// TIA Portal V21 export
FUNCTION "T_PausaLavoro" : Void   // FC81, LAD
{ S7_Optimized_Access := 'TRUE' }
// stored: SetENOAutomatically false
   VAR_IN_OUT
      PausaLavoro : "Std_PausaLavoro";
   END_VAR
   VAR_TEMP   // added for the SCL form of the ladder/FBD networks
      _w1 : Bool;
   END_VAR
BEGIN

REGION Network 1
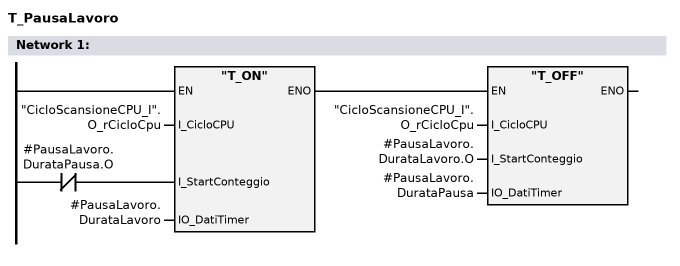
   RUNG wire#powerrail
      "T_ON"(I_StartConteggio := wire#w1, I_CicloCPU := "CicloScansioneCPU_I".O_rCicloCpu, IO_DatiTimer := #PausaLavoro.DurataLavoro)
      "T_OFF"(I_CicloCPU := "CicloScansioneCPU_I".O_rCicloCpu, I_StartConteggio := #PausaLavoro.DurataLavoro.O, IO_DatiTimer := #PausaLavoro.DurataPausa)
   END_RUNG
   RUNG wire#powerrail
      I_Contact( #PausaLavoro.DurataPausa.O )
   END_RUNG wire#w1
   // the same network as SCL:
   "T_ON"(I_CicloCPU := "CicloScansioneCPU_I".O_rCicloCpu,
          I_StartConteggio := NOT #PausaLavoro.DurataPausa.O,
          IO_DatiTimer := #PausaLavoro.DurataLavoro,
          ENO => #_w1);
   IF #_w1 THEN
       "T_OFF"(I_CicloCPU := "CicloScansioneCPU_I".O_rCicloCpu,
               I_StartConteggio := #PausaLavoro.DurataLavoro.O,
               IO_DatiTimer := #PausaLavoro.DurataPausa);
   END_IF;
END_REGION

REGION Network 2 (SCL)
   ENO := NOT #PausaLavoro.DurataPausa.O OR NOT #PausaLavoro.Abilitazione;
END_REGION
END_FUNCTION
